TYPE DUT_HMI_13_MANUALS :
STRUCT
	PS : ARRAY[0..CNC.NUM_MAX_MANUALS_13-1] OF BOOL;
	LS : ARRAY[0..CNC.NUM_MAX_MANUALS_13-1] OF BOOL;
END_STRUCT
END_TYPE

(* stored: Version 1.1.0.1, ProductVersion 3.1.4024.13
   DUT DUT_HMI_13_MANUALS: Id {8e653139-ec9b-43bc-95fd-d594a743efb2} *)
